// TIA Portal project "Banda_Asamblare" (V15.1)

(* hardware
DEVICE "S71500/ET200MP station_1"  S7-1500 station
   slot 0: "Rail_0"  Rack  6ES7 590-1***0-0AA0
   slot 1: "PLC_1"  CPU 1513-1 PN  6ES7 513-1AL02-0AB0  V2.6
      slot 3: "CPU display_1"  6ES7591-1AA00-0AA0
*)

// ===== PLC "PLC_1"  CPU 1513-1 PN =====

VAR_GLOBAL   // PLC tag table "Default tag table"
   "Clock_Byte" AT %MB0 : Byte;
   "Clock_10Hz" AT %M0.0 : Bool;
   "Clock_5Hz" AT %M0.1 : Bool;
   "Clock_2.5Hz" AT %M0.2 : Bool;
   "Clock_2Hz" AT %M0.3 : Bool;
   "Clock_1.25Hz" AT %M0.4 : Bool;
   "Clock_1Hz" AT %M0.5 : Bool;
   "Clock_0.625Hz" AT %M0.6 : Bool;
   "Clock_0.5Hz" AT %M0.7 : Bool;
END_VAR

DATA_BLOCK "Alarme"   // DB1
{ S7_Optimized_Access := 'TRUE' }
VERSION : 0.1
   VAR
      alarme_vect : Array[0..15] of Bool;
      alarme_gather : Word;
   END_VAR
BEGIN
END_DATA_BLOCK

DATA_BLOCK "Avarii"   // DB2
{ S7_Optimized_Access := 'TRUE' }
VERSION : 0.1
   VAR
      avarie_start : Bool;
      avarie_cuptor : Bool;
      avarie_aplatizor : Bool;
      avarie_forme : Bool;
      avarie_taiere : Bool;
      avarie_curatare : Bool;
      avarie_general : Bool;
      container1_plin : Bool;
      container2_plin : Bool;
      container3_plin : Bool;
      container_plin_general : Bool;
      limite_containere : Bool;
   END_VAR
BEGIN
END_DATA_BLOCK

DATA_BLOCK "Mecanisme"   // DB3
{ S7_Optimized_Access := 'TRUE' }
VERSION : 0.1
   VAR
      block_start : Bool;
      punere_block_material : Bool;
      cuptor : Bool;
      temperatura_cuptor : Real;
      "temperatura dorita la cuptor" : Real;
      temp_dorita_atinsa : Bool;
      aplatizor : Bool;
      forma : UInt;
      ajuns_la_forma1 : Bool;
      ajuns_la_forma2 : Bool;
      ajuns_la_forma3 : Bool;
      taiere1 : Bool;
      taiere2 : Bool;
      taiere3 : Bool;
      curatare1 : Bool;
      curatare2 : Bool;
      curatare3 : Bool;
      container_f1 : UInt;
      container_f2 : UInt;
      container_f3 : UInt;
      servo : UInt;
      limita_c1 : UInt;
      limita_c2 : UInt;
      limita_c3 : UInt;
      cond_cuptor : Bool;
   END_VAR
BEGIN
END_DATA_BLOCK

DATA_BLOCK "Butoane"   // DB4
{ S7_Optimized_Access := 'TRUE' }
VERSION : 0.1
   VAR
      btn_start : Bool;
      btn_esd : Bool;
      btn_stop : Bool;
      reset_esd : Bool;
      pornire : Bool;
      esd : Bool;
      "blocare_start_pe timer" : Bool;
      mentinere_timer_punere_material : Bool;
      "reset avarii" : Bool;
      timer_oprit : Bool;
      golire_c1 : Bool;
      golire_c2 : Bool;
      golire_c3 : Bool;
   END_VAR
BEGIN
END_DATA_BLOCK

DATA_BLOCK "Benzi"   // DB5
{ S7_Optimized_Access := 'TRUE' }
VERSION : 0.1
   VAR
      plecat_b1 : Bool;
      plecat_b2 : Bool;
      plecat_b3 : Bool;
      plecat_b41 : Bool;
      plecat_b42 : Bool;
      plecat_b43 : Bool;
      plecat_b51 : Bool;
      plecat_b52 : Bool;
      plecat_b53 : Bool;
      plecat_b61 : Bool;
      plecat_b62 : Bool;
      plecat_b63 : Bool;
   END_VAR
BEGIN
END_DATA_BLOCK

DATA_BLOCK "Comenzi_DB"   // DB7
{ S7_Optimized_Access := 'TRUE' }
VERSION : 0.1
// stored: InstanceOfName Comenzi
"Comenzi"
BEGIN
END_DATA_BLOCK

DATA_BLOCK "rising edges"   // DB9
{ S7_Optimized_Access := 'TRUE' }
VERSION : 0.1
   VAR
      re1 : Bool;
      re2 : Bool;
      re3 : Bool;
      re4 : Bool;
      re5 : Bool;
      re6 : Bool;
      re7 : Bool;
      re8 : Bool;
   END_VAR
BEGIN
END_DATA_BLOCK

DATA_BLOCK "Simulare_DB"   // DB13
{ S7_Optimized_Access := 'TRUE' }
VERSION : 0.1
// stored: InstanceOfName Simulare
"Simulare"
BEGIN
END_DATA_BLOCK

// folder: System blocks/Program resources

DATA_BLOCK "reset esd"   // DB6
{ S7_Optimized_Access := 'TRUE' }
AUTHOR : Simatic
FAMILY : IEC
NAME : IEC_TMR
VERSION : 1.0
// stored: InstanceOfName IEC_TIMER
"IEC_TIMER"
BEGIN
END_DATA_BLOCK

// folder: (top level)

FUNCTION_BLOCK "Simulare"   // FB1, LAD
{ S7_Optimized_Access := 'TRUE' }
VERSION : 0.1
   VAR_INPUT
      btn_pornire : Bool;
      b1_plecat : Bool;
      b2_plecat : Bool;
      b3_plecat : Bool;
      b41_plecat : Bool;
      b42_plecat : Bool;
      b43_plecat : Bool;
      b51_plecat : Bool;
      b52_plecat : Bool;
      b53_plecat : Bool;
      b61_plecat : Bool;
      b62_plecat : Bool;
      b63_plecat : Bool;
      cond_cuptor : Bool;
      forma : UInt;
   END_VAR
   VAR_OUTPUT
      cuptor_pornit : Bool;
      aplatizor_pornit : Bool;
      forma1 : Bool;
      forma2 : Bool;
      forma3 : Bool;
      taiere1 : Bool;
      taiere2 : Bool;
      taiere3 : Bool;
      curatare1 : Bool;
      curatare2 : Bool;
      curatare3 : Bool;
      container1 : UInt;
      container2 : UInt;
      container3 : UInt;
      servo : UInt;
   END_VAR
   VAR_IN_OUT
      pune_material : Bool;
      btn_golire1 : Bool;
      btn_golire2 : Bool;
      btn_golire3 : Bool;
      temp_cuptor : Real;
   END_VAR
   VAR
      re1 : Bool;
      re2 : Bool;
      re3 : Bool;
      re4 : Bool;
      re5 : Bool;
      "timer reset punere material" : TON_TIME;
      mentinere_timer_material : Bool;
      timer_aplatizare : TON_TIME;
      "tiimer forma" : TON_TIME;
      "timer taiere1" : TON_TIME;
      "timer taiere2" : TON_TIME;
      "timer taiere3" : TON_TIME;
      "timer curatare1" : TON_TIME;
      "timer curatare 2" : TON_TIME;
      "timer curatare 3" : TON_TIME;
      "reset golire1" : TON_TIME;
      "reset golire 2" : TON_TIME;
      "reset golire 3" : TON_TIME;
   END_VAR
   VAR_TEMP   // added for the SCL form of the ladder/FBD networks
      _w1 : Bool;
      _w2 : Bool;
      _w3 : Bool;
   END_VAR
BEGIN

REGION Network 1: pune un block de material pe banda
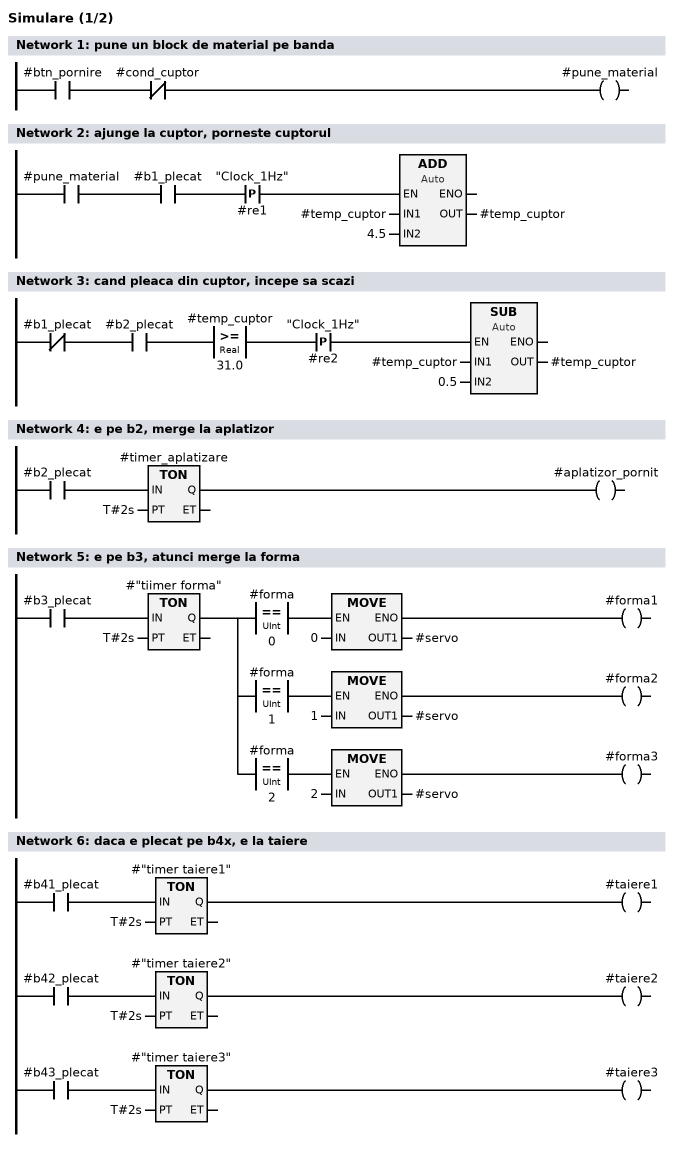
   RUNG wire#powerrail
      Contact( #btn_pornire )
      I_Contact( #cond_cuptor )
      Coil( #pune_material )
   END_RUNG
   // the same network as SCL:
   #pune_material := #btn_pornire AND NOT #cond_cuptor;
END_REGION

REGION Network 2: ajunge la cuptor, porneste cuptorul
   RUNG wire#powerrail
      Contact( #pune_material )
      Contact( #b1_plecat )
      P_Contact(operand := "Clock_1Hz", bit := #re1)
      Add(in1 := #temp_cuptor, in2 := 4.5, out => #temp_cuptor)
   END_RUNG
   // the same network as SCL:
   #_w1 := #pune_material AND #b1_plecat AND "Clock_1Hz" AND NOT #re1;   // rising edge of "Clock_1Hz"
   #re1 := "Clock_1Hz";
   IF #_w1 THEN #temp_cuptor := #temp_cuptor + 4.5; END_IF;
END_REGION

REGION Network 3: cand pleaca din cuptor, incepe sa scazi
   RUNG wire#powerrail
      I_Contact( #b1_plecat )
      Contact( #b2_plecat )
      { S7_Templates := "SrcType := Real" } GE_Contact(in1 := #temp_cuptor, in2 := 31.0)
      P_Contact(operand := "Clock_1Hz", bit := #re2)
      Sub(in1 := #temp_cuptor, in2 := 0.5, out => #temp_cuptor)
   END_RUNG
   // the same network as SCL:
   #_w1 := NOT #b1_plecat AND #b2_plecat AND (#temp_cuptor >= 31.0) AND "Clock_1Hz" AND NOT #re2;   // rising edge of "Clock_1Hz"
   #re2 := "Clock_1Hz";
   IF #_w1 THEN #temp_cuptor := #temp_cuptor - 0.5; END_IF;
END_REGION

REGION Network 4: e pe b2, merge la aplatizor
   #timer_aplatizare(IN := #b2_plecat, PT := T#2s);   // TON
   #aplatizor_pornit := #timer_aplatizare.Q;
END_REGION

REGION Network 5: e pe b3, atunci merge la forma
   #"tiimer forma"(IN := #b3_plecat, PT := T#2s);   // TON
   #_w1 := #"tiimer forma".Q AND (#forma = 0);
   IF #_w1 THEN #servo := 0; END_IF;
   #forma1 := #_w1;
   #_w2 := #"tiimer forma".Q AND (#forma = 1);
   IF #_w2 THEN #servo := 1; END_IF;
   #forma2 := #_w2;
   #_w3 := #"tiimer forma".Q AND (#forma = 2);
   IF #_w3 THEN #servo := 2; END_IF;
   #forma3 := #_w3;
END_REGION

REGION Network 6: daca e plecat pe b4x, e la taiere
   #"timer taiere1"(IN := #b41_plecat, PT := T#2s);   // TON
   #taiere1 := #"timer taiere1".Q;
   #"timer taiere2"(IN := #b42_plecat, PT := T#2s);   // TON
   #taiere2 := #"timer taiere2".Q;
   #"timer taiere3"(IN := #b43_plecat, PT := T#2s);   // TON
   #taiere3 := #"timer taiere3".Q;
END_REGION

REGION Network 7: daca e pe banda b5x, sa dea drumul la curatari
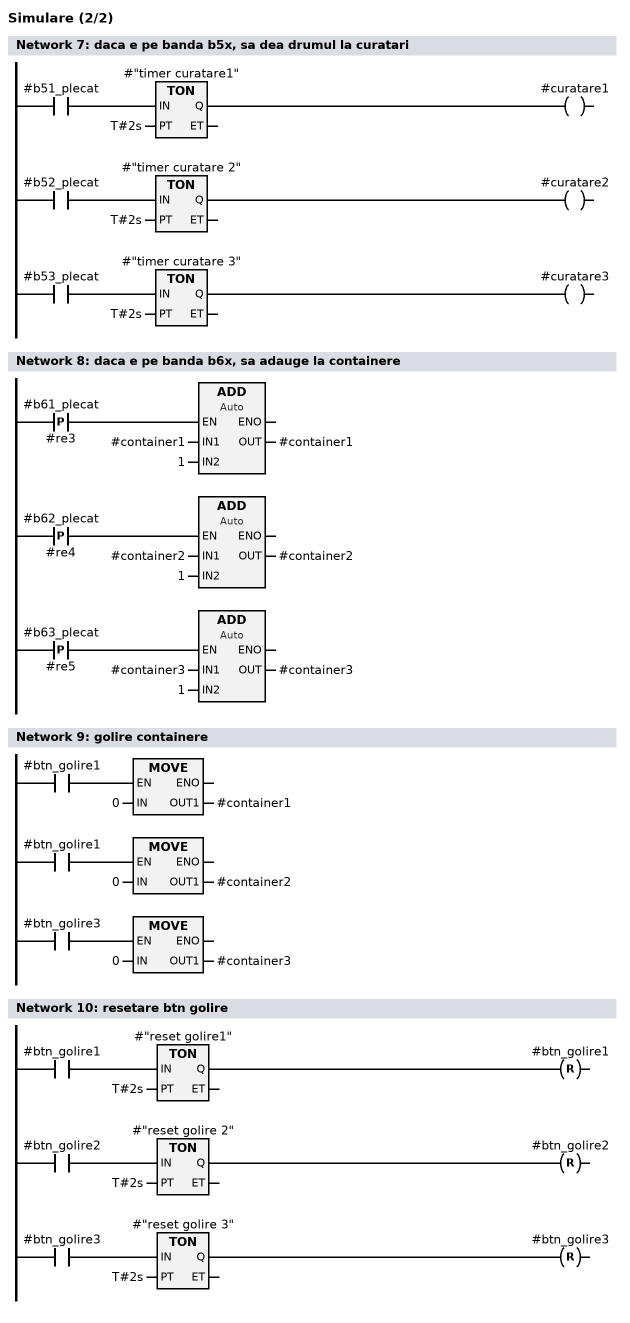
   #"timer curatare1"(IN := #b51_plecat, PT := T#2s);   // TON
   #curatare1 := #"timer curatare1".Q;
   #"timer curatare 2"(IN := #b52_plecat, PT := T#2s);   // TON
   #curatare2 := #"timer curatare 2".Q;
   #"timer curatare 3"(IN := #b53_plecat, PT := T#2s);   // TON
   #curatare3 := #"timer curatare 3".Q;
END_REGION

REGION Network 8: daca e pe banda b6x, sa adauge la containere
   RUNG wire#powerrail
      P_Contact(operand := #b61_plecat, bit := #re3)
      Add(in1 := #container1, in2 := 1, out => #container1)
   END_RUNG
   RUNG wire#powerrail
      P_Contact(operand := #b62_plecat, bit := #re4)
      Add(in1 := #container2, in2 := 1, out => #container2)
   END_RUNG
   RUNG wire#powerrail
      P_Contact(operand := #b63_plecat, bit := #re5)
      Add(in1 := #container3, in2 := 1, out => #container3)
   END_RUNG
   // the same network as SCL:
   #_w1 := #b61_plecat AND NOT #re3;   // rising edge of #b61_plecat
   #re3 := #b61_plecat;
   IF #_w1 THEN #container1 := #container1 + 1; END_IF;
   #_w2 := #b62_plecat AND NOT #re4;   // rising edge of #b62_plecat
   #re4 := #b62_plecat;
   IF #_w2 THEN #container2 := #container2 + 1; END_IF;
   #_w3 := #b63_plecat AND NOT #re5;   // rising edge of #b63_plecat
   #re5 := #b63_plecat;
   IF #_w3 THEN #container3 := #container3 + 1; END_IF;
END_REGION

REGION Network 9: golire containere
   RUNG wire#powerrail
      Contact( #btn_golire1 )
      Move(in := 0, out1 => #container1)
   END_RUNG
   RUNG wire#powerrail
      Contact( #btn_golire1 )
      Move(in := 0, out1 => #container2)
   END_RUNG
   RUNG wire#powerrail
      Contact( #btn_golire3 )
      Move(in := 0, out1 => #container3)
   END_RUNG
   // the same network as SCL:
   IF #btn_golire1 THEN
       #container1 := 0;
       #container2 := 0;
   END_IF;
   IF #btn_golire3 THEN #container3 := 0; END_IF;
END_REGION

REGION Network 10: resetare btn golire
   #"reset golire1"(IN := #btn_golire1, PT := T#2s);   // TON
   IF #"reset golire1".Q THEN #btn_golire1 := FALSE; END_IF;
   #"reset golire 2"(IN := #btn_golire2, PT := T#2s);   // TON
   IF #"reset golire 2".Q THEN #btn_golire2 := FALSE; END_IF;
   #"reset golire 3"(IN := #btn_golire3, PT := T#2s);   // TON
   IF #"reset golire 3".Q THEN #btn_golire3 := FALSE; END_IF;
END_REGION
END_FUNCTION_BLOCK

FUNCTION_BLOCK "Comenzi"   // FB2, LAD
{ S7_Optimized_Access := 'TRUE' }
VERSION : 0.1
   VAR_INPUT
      temp_cuptor : Real;
      temp_dorita : Real;
      pune_material : Bool;
      aplatizor_pornit : Bool;
      forma1 : Bool;
      forma2 : Bool;
      forma3 : Bool;
      taiere1 : Bool;
      taiere2 : Bool;
      taiere3 : Bool;
      curatare1 : Bool;
      curatare2 : Bool;
      curatare3 : Bool;
   END_VAR
   VAR_OUTPUT
      b1_plecat : Bool;
      b2_plecat : Bool;
      b3_plecat : Bool;
      b41_plecat : Bool;
      b42_plecat : Bool;
      b43_plecat : Bool;
      b51_plecat : Bool;
      b52_plecat : Bool;
      b53_plecat : Bool;
      b61_plecat : Bool;
      b62_plecat : Bool;
      b63_plecat : Bool;
      cond_cuptor : Bool;
   END_VAR
   VAR
      "timer plecare b1" : TON_TIME;
      incc : Int;
      edg : Bool;
   END_VAR
BEGIN

REGION Network 1: pleaca spre cuptor
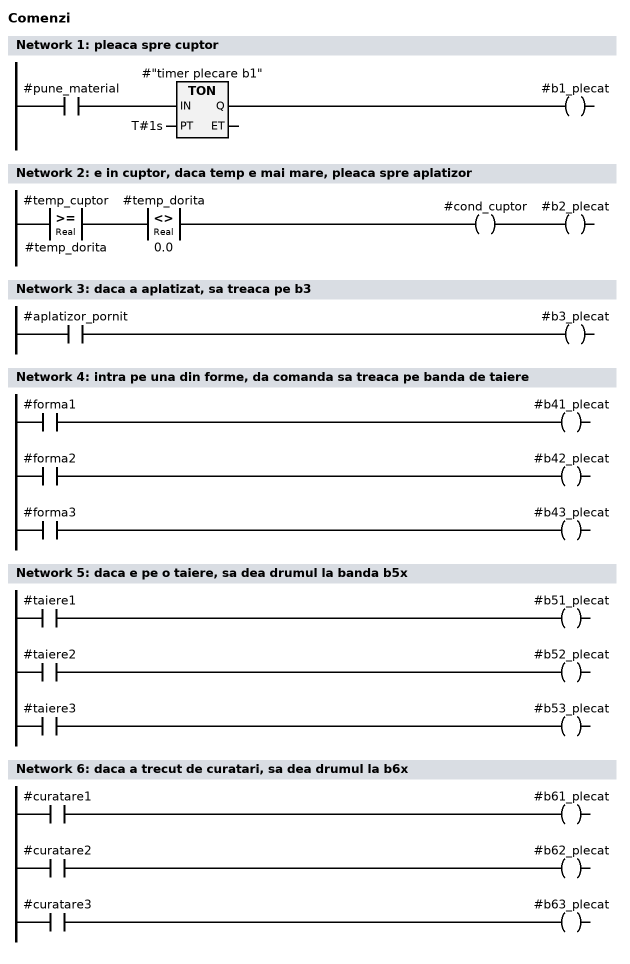
   #"timer plecare b1"(IN := #pune_material, PT := T#1s);   // TON
   #b1_plecat := #"timer plecare b1".Q;
END_REGION

REGION Network 2: e in cuptor, daca temp e mai mare, pleaca spre aplatizor
   RUNG wire#powerrail
      { S7_Templates := "SrcType := Real" } GE_Contact(in1 := #temp_cuptor, in2 := #temp_dorita)
      { S7_Templates := "SrcType := Real" } NE_Contact(in1 := #temp_dorita, in2 := 0.0)
      Coil( #cond_cuptor )
      Coil( #b2_plecat )
   END_RUNG
   // the same network as SCL:
   #cond_cuptor := (#temp_cuptor >= #temp_dorita) AND (#temp_dorita <> 0.0);
   #b2_plecat := #cond_cuptor;
END_REGION

REGION Network 3: daca a aplatizat, sa treaca pe b3
   RUNG wire#powerrail
      Contact( #aplatizor_pornit )
      Coil( #b3_plecat )
   END_RUNG
   // the same network as SCL:
   #b3_plecat := #aplatizor_pornit;
END_REGION

REGION Network 4: intra pe una din forme, da comanda sa treaca pe banda de taiere
   RUNG wire#powerrail
      Contact( #forma1 )
      Coil( #b41_plecat )
   END_RUNG
   RUNG wire#powerrail
      Contact( #forma2 )
      Coil( #b42_plecat )
   END_RUNG
   RUNG wire#powerrail
      Contact( #forma3 )
      Coil( #b43_plecat )
   END_RUNG
   // the same network as SCL:
   #b41_plecat := #forma1;
   #b42_plecat := #forma2;
   #b43_plecat := #forma3;
END_REGION

REGION Network 5: daca e pe o taiere, sa dea drumul la banda b5x
   RUNG wire#powerrail
      Contact( #taiere1 )
      Coil( #b51_plecat )
   END_RUNG
   RUNG wire#powerrail
      Contact( #taiere2 )
      Coil( #b52_plecat )
   END_RUNG
   RUNG wire#powerrail
      Contact( #taiere3 )
      Coil( #b53_plecat )
   END_RUNG
   // the same network as SCL:
   #b51_plecat := #taiere1;
   #b52_plecat := #taiere2;
   #b53_plecat := #taiere3;
END_REGION

REGION Network 6: daca a trecut de curatari, sa dea drumul la b6x
   RUNG wire#powerrail
      Contact( #curatare1 )
      Coil( #b61_plecat )
   END_RUNG
   RUNG wire#powerrail
      Contact( #curatare2 )
      Coil( #b62_plecat )
   END_RUNG
   RUNG wire#powerrail
      Contact( #curatare3 )
      Coil( #b63_plecat )
   END_RUNG
   // the same network as SCL:
   #b61_plecat := #curatare1;
   #b62_plecat := #curatare2;
   #b63_plecat := #curatare3;
END_REGION
END_FUNCTION_BLOCK

ORGANIZATION_BLOCK "Main"   // OB1, LAD, ProgramCycle
TITLE = "Main Program Sweep (Cycle)"
{ S7_Optimized_Access := 'TRUE' }
VERSION : 0.1
   VAR_INPUT
      Initial_Call : Bool;   // Initial call of this OB
      Remanence : Bool;   // =True, if remanent data are available
   END_VAR
BEGIN

REGION Network 1: buton start
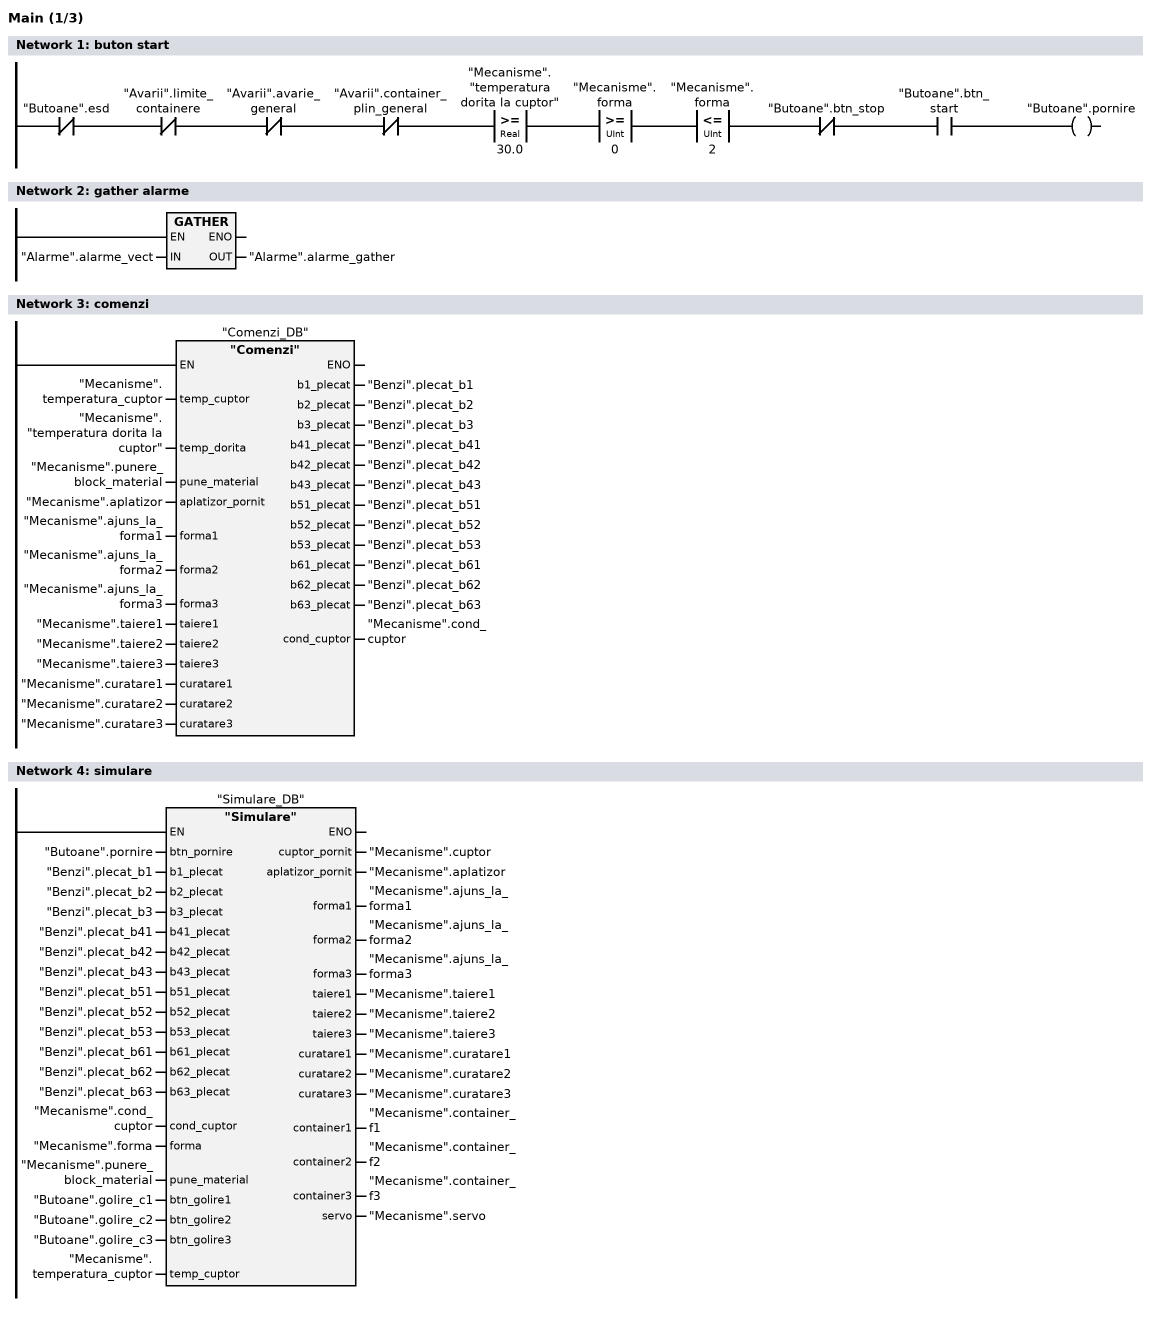
   RUNG wire#powerrail
      I_Contact( "Butoane".esd )
      I_Contact( "Avarii".limite_containere )
      I_Contact( "Avarii".avarie_general )
      I_Contact( "Avarii".container_plin_general )
      { S7_Templates := "SrcType := Real" } GE_Contact(in1 := "Mecanisme"."temperatura dorita la cuptor", in2 := 30.0)
      { S7_Templates := "SrcType := UInt" } GE_Contact(in1 := "Mecanisme".forma, in2 := 0)
      { S7_Templates := "SrcType := UInt" } LE_Contact(in1 := "Mecanisme".forma, in2 := 2)
      I_Contact( "Butoane".btn_stop )
      Contact( "Butoane".btn_start )
      Coil( "Butoane".pornire )
   END_RUNG
   // the same network as SCL:
   "Butoane".pornire := NOT "Butoane".esd AND NOT "Avarii".limite_containere AND NOT "Avarii".avarie_general AND NOT "Avarii".container_plin_general AND ("Mecanisme"."temperatura dorita la cuptor" >= 30.0) AND ("Mecanisme".forma >= 0) AND ("Mecanisme".forma <= 2) AND NOT "Butoane".btn_stop AND "Butoane".btn_start;
END_REGION

REGION Network 2: gather alarme
   GATHER(IN := "Alarme".alarme_vect, OUT => "Alarme".alarme_gather);
END_REGION

REGION Network 3: comenzi
   RUNG wire#powerrail
      "Comenzi_DB"(temp_cuptor := "Mecanisme".temperatura_cuptor, temp_dorita := "Mecanisme"."temperatura dorita la cuptor", pune_material := "Mecanisme".punere_block_material, aplatizor_pornit := "Mecanisme".aplatizor, forma1 := "Mecanisme".ajuns_la_forma1, forma2 := "Mecanisme".ajuns_la_forma2, forma3 := "Mecanisme".ajuns_la_forma3, taiere1 := "Mecanisme".taiere1, taiere2 := "Mecanisme".taiere2, taiere3 := "Mecanisme".taiere3, curatare1 := "Mecanisme".curatare1, curatare2 := "Mecanisme".curatare2, curatare3 := "Mecanisme".curatare3, b1_plecat => "Benzi".plecat_b1, b2_plecat => "Benzi".plecat_b2, b3_plecat => "Benzi".plecat_b3, b41_plecat => "Benzi".plecat_b41, b42_plecat => "Benzi".plecat_b42, b43_plecat => "Benzi".plecat_b43, b51_plecat => "Benzi".plecat_b51, b52_plecat => "Benzi".plecat_b52, b53_plecat => "Benzi".plecat_b53, b61_plecat => "Benzi".plecat_b61, b62_plecat => "Benzi".plecat_b62, b63_plecat => "Benzi".plecat_b63, cond_cuptor => "Mecanisme".cond_cuptor)
   END_RUNG
   // the same network as SCL:
   "Comenzi_DB"(temp_cuptor := "Mecanisme".temperatura_cuptor,   // "Comenzi"
                temp_dorita := "Mecanisme"."temperatura dorita la cuptor",
                pune_material := "Mecanisme".punere_block_material,
                aplatizor_pornit := "Mecanisme".aplatizor,
                forma1 := "Mecanisme".ajuns_la_forma1,
                forma2 := "Mecanisme".ajuns_la_forma2,
                forma3 := "Mecanisme".ajuns_la_forma3,
                taiere1 := "Mecanisme".taiere1,
                taiere2 := "Mecanisme".taiere2,
                taiere3 := "Mecanisme".taiere3,
                curatare1 := "Mecanisme".curatare1,
                curatare2 := "Mecanisme".curatare2,
                curatare3 := "Mecanisme".curatare3,
                b1_plecat => "Benzi".plecat_b1,
                b2_plecat => "Benzi".plecat_b2,
                b3_plecat => "Benzi".plecat_b3,
                b41_plecat => "Benzi".plecat_b41,
                b42_plecat => "Benzi".plecat_b42,
                b43_plecat => "Benzi".plecat_b43,
                b51_plecat => "Benzi".plecat_b51,
                b52_plecat => "Benzi".plecat_b52,
                b53_plecat => "Benzi".plecat_b53,
                b61_plecat => "Benzi".plecat_b61,
                b62_plecat => "Benzi".plecat_b62,
                b63_plecat => "Benzi".plecat_b63,
                cond_cuptor => "Mecanisme".cond_cuptor);
END_REGION

REGION Network 4: simulare
   RUNG wire#powerrail
      "Simulare_DB"(btn_pornire := "Butoane".pornire, b1_plecat := "Benzi".plecat_b1, b2_plecat := "Benzi".plecat_b2, b3_plecat := "Benzi".plecat_b3, b41_plecat := "Benzi".plecat_b41, b42_plecat := "Benzi".plecat_b42, b43_plecat := "Benzi".plecat_b43, b51_plecat := "Benzi".plecat_b51, b52_plecat := "Benzi".plecat_b52, b53_plecat := "Benzi".plecat_b53, b61_plecat := "Benzi".plecat_b61, b62_plecat := "Benzi".plecat_b62, b63_plecat := "Benzi".plecat_b63, cond_cuptor := "Mecanisme".cond_cuptor, forma := "Mecanisme".forma, btn_golire1 := "Butoane".golire_c1, btn_golire2 := "Butoane".golire_c2, btn_golire3 := "Butoane".golire_c3, pune_material := "Mecanisme".punere_block_material, temp_cuptor := "Mecanisme".temperatura_cuptor, cuptor_pornit => "Mecanisme".cuptor, aplatizor_pornit => "Mecanisme".aplatizor, forma1 => "Mecanisme".ajuns_la_forma1, forma2 => "Mecanisme".ajuns_la_forma2, forma3 => "Mecanisme".ajuns_la_forma3, taiere1 => "Mecanisme".taiere1, taiere2 => "Mecanisme".taiere2, taiere3 => "Mecanisme".taiere3, curatare1 => "Mecanisme".curatare1, curatare2 => "Mecanisme".curatare2, curatare3 => "Mecanisme".curatare3, container1 => "Mecanisme".container_f1, container2 => "Mecanisme".container_f2, container3 => "Mecanisme".container_f3, servo => "Mecanisme".servo)
   END_RUNG
   // the same network as SCL:
   "Simulare_DB"(btn_pornire := "Butoane".pornire,   // "Simulare"
                 b1_plecat := "Benzi".plecat_b1,
                 b2_plecat := "Benzi".plecat_b2,
                 b3_plecat := "Benzi".plecat_b3,
                 b41_plecat := "Benzi".plecat_b41,
                 b42_plecat := "Benzi".plecat_b42,
                 b43_plecat := "Benzi".plecat_b43,
                 b51_plecat := "Benzi".plecat_b51,
                 b52_plecat := "Benzi".plecat_b52,
                 b53_plecat := "Benzi".plecat_b53,
                 b61_plecat := "Benzi".plecat_b61,
                 b62_plecat := "Benzi".plecat_b62,
                 b63_plecat := "Benzi".plecat_b63,
                 cond_cuptor := "Mecanisme".cond_cuptor,
                 forma := "Mecanisme".forma,
                 pune_material := "Mecanisme".punere_block_material,
                 btn_golire1 := "Butoane".golire_c1,
                 btn_golire2 := "Butoane".golire_c2,
                 btn_golire3 := "Butoane".golire_c3,
                 temp_cuptor := "Mecanisme".temperatura_cuptor,
                 cuptor_pornit => "Mecanisme".cuptor,
                 aplatizor_pornit => "Mecanisme".aplatizor,
                 forma1 => "Mecanisme".ajuns_la_forma1,
                 forma2 => "Mecanisme".ajuns_la_forma2,
                 forma3 => "Mecanisme".ajuns_la_forma3,
                 taiere1 => "Mecanisme".taiere1,
                 taiere2 => "Mecanisme".taiere2,
                 taiere3 => "Mecanisme".taiere3,
                 curatare1 => "Mecanisme".curatare1,
                 curatare2 => "Mecanisme".curatare2,
                 curatare3 => "Mecanisme".curatare3,
                 container1 => "Mecanisme".container_f1,
                 container2 => "Mecanisme".container_f2,
                 container3 => "Mecanisme".container_f3,
                 servo => "Mecanisme".servo);
END_REGION

REGION Network 5: esd
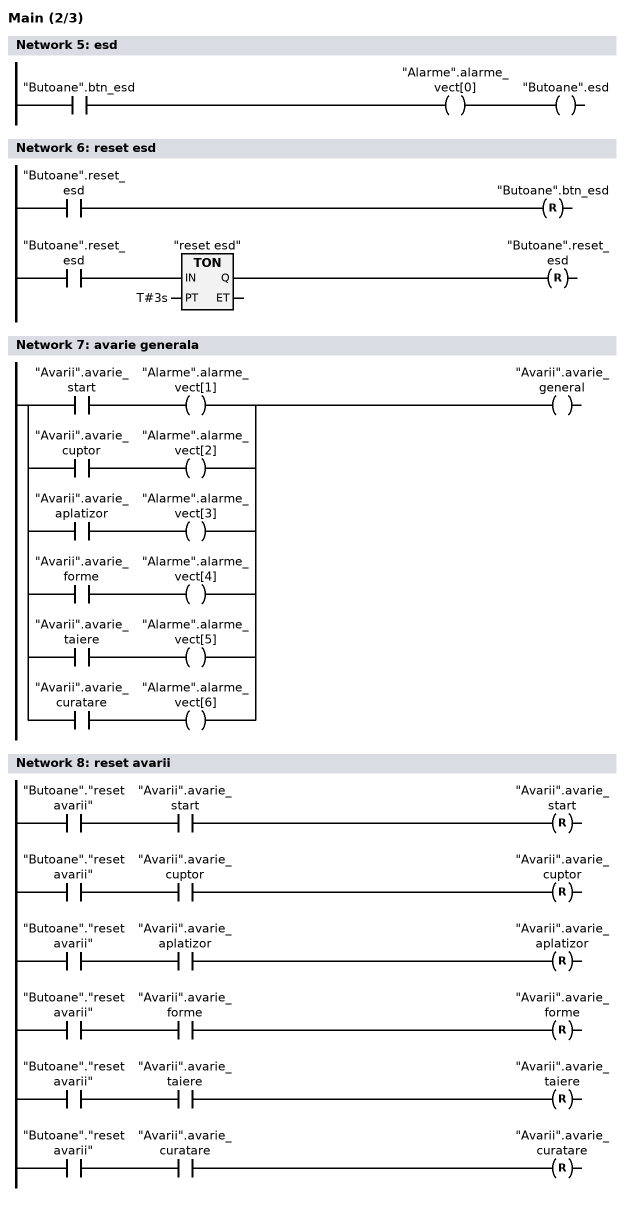
   RUNG wire#powerrail
      Contact( "Butoane".btn_esd )
      Coil( "Alarme".alarme_vect[0] )
      Coil( "Butoane".esd )
   END_RUNG
   // the same network as SCL:
   "Alarme".alarme_vect[0] := "Butoane".btn_esd;
   "Butoane".esd := "Butoane".btn_esd;
END_REGION

REGION Network 6: reset esd
   IF "Butoane".reset_esd THEN "Butoane".btn_esd := FALSE; END_IF;
   "reset esd".TON(IN := "Butoane".reset_esd, PT := T#3s);
   IF "reset esd".Q THEN "Butoane".reset_esd := FALSE; END_IF;
END_REGION

REGION Network 7: avarie generala
   RUNG wire#powerrail
      Contact( "Avarii".avarie_start )
      Coil( "Alarme".alarme_vect[1] )
      wire#w1
      Coil( "Avarii".avarie_general )
   END_RUNG
   RUNG wire#powerrail
      Contact( "Avarii".avarie_cuptor )
      Coil( "Alarme".alarme_vect[2] )
   END_RUNG wire#w1
   RUNG wire#powerrail
      Contact( "Avarii".avarie_aplatizor )
      Coil( "Alarme".alarme_vect[3] )
   END_RUNG wire#w1
   RUNG wire#powerrail
      Contact( "Avarii".avarie_forme )
      Coil( "Alarme".alarme_vect[4] )
   END_RUNG wire#w1
   RUNG wire#powerrail
      Contact( "Avarii".avarie_taiere )
      Coil( "Alarme".alarme_vect[5] )
   END_RUNG wire#w1
   RUNG wire#powerrail
      Contact( "Avarii".avarie_curatare )
      Coil( "Alarme".alarme_vect[6] )
   END_RUNG wire#w1
   // the same network as SCL:
   "Alarme".alarme_vect[1] := "Avarii".avarie_start;
   "Alarme".alarme_vect[2] := "Avarii".avarie_cuptor;
   "Alarme".alarme_vect[3] := "Avarii".avarie_aplatizor;
   "Alarme".alarme_vect[4] := "Avarii".avarie_forme;
   "Alarme".alarme_vect[5] := "Avarii".avarie_taiere;
   "Alarme".alarme_vect[6] := "Avarii".avarie_curatare;
   "Avarii".avarie_general := "Avarii".avarie_start OR "Avarii".avarie_cuptor OR "Avarii".avarie_aplatizor OR "Avarii".avarie_forme OR "Avarii".avarie_taiere OR "Avarii".avarie_curatare;
END_REGION

REGION Network 8: reset avarii
   RUNG wire#powerrail
      Contact( "Butoane"."reset avarii" )
      Contact( "Avarii".avarie_start )
      R_Coil( "Avarii".avarie_start )
   END_RUNG
   RUNG wire#powerrail
      Contact( "Butoane"."reset avarii" )
      Contact( "Avarii".avarie_cuptor )
      R_Coil( "Avarii".avarie_cuptor )
   END_RUNG
   RUNG wire#powerrail
      Contact( "Butoane"."reset avarii" )
      Contact( "Avarii".avarie_aplatizor )
      R_Coil( "Avarii".avarie_aplatizor )
   END_RUNG
   RUNG wire#powerrail
      Contact( "Butoane"."reset avarii" )
      Contact( "Avarii".avarie_forme )
      R_Coil( "Avarii".avarie_forme )
   END_RUNG
   RUNG wire#powerrail
      Contact( "Butoane"."reset avarii" )
      Contact( "Avarii".avarie_taiere )
      R_Coil( "Avarii".avarie_taiere )
   END_RUNG
   RUNG wire#powerrail
      Contact( "Butoane"."reset avarii" )
      Contact( "Avarii".avarie_curatare )
      R_Coil( "Avarii".avarie_curatare )
   END_RUNG
   // the same network as SCL:
   IF "Butoane"."reset avarii" AND "Avarii".avarie_start THEN "Avarii".avarie_start := FALSE; END_IF;
   IF "Butoane"."reset avarii" AND "Avarii".avarie_cuptor THEN "Avarii".avarie_cuptor := FALSE; END_IF;
   IF "Butoane"."reset avarii" AND "Avarii".avarie_aplatizor THEN "Avarii".avarie_aplatizor := FALSE; END_IF;
   IF "Butoane"."reset avarii" AND "Avarii".avarie_forme THEN "Avarii".avarie_forme := FALSE; END_IF;
   IF "Butoane"."reset avarii" AND "Avarii".avarie_taiere THEN "Avarii".avarie_taiere := FALSE; END_IF;
   IF "Butoane"."reset avarii" AND "Avarii".avarie_curatare THEN "Avarii".avarie_curatare := FALSE; END_IF;
END_REGION

REGION Network 9: container plin general
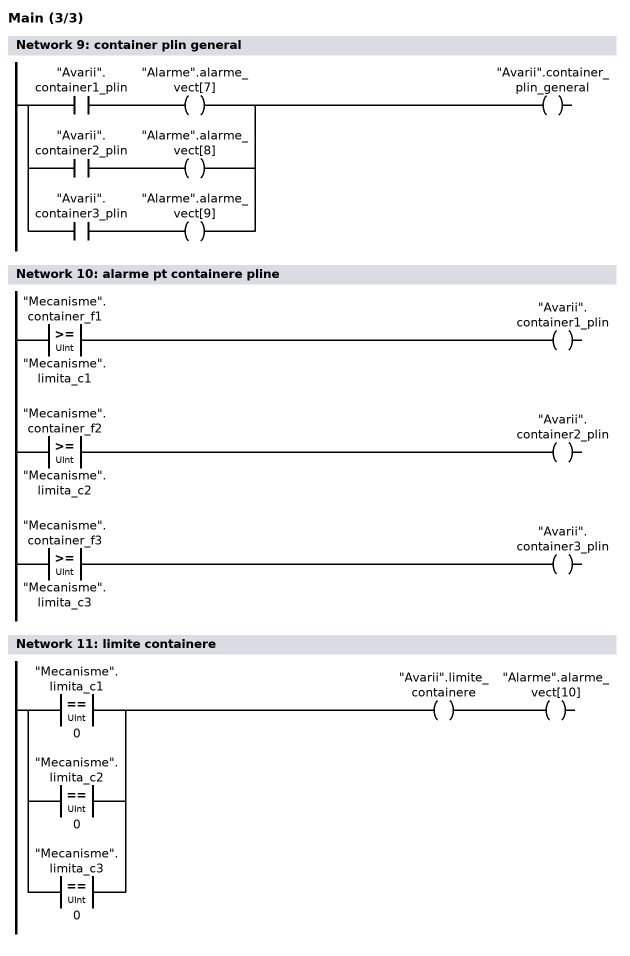
   RUNG wire#powerrail
      Contact( "Avarii".container1_plin )
      Coil( "Alarme".alarme_vect[7] )
      wire#w1
      Coil( "Avarii".container_plin_general )
   END_RUNG
   RUNG wire#powerrail
      Contact( "Avarii".container2_plin )
      Coil( "Alarme".alarme_vect[8] )
   END_RUNG wire#w1
   RUNG wire#powerrail
      Contact( "Avarii".container3_plin )
      Coil( "Alarme".alarme_vect[9] )
   END_RUNG wire#w1
   // the same network as SCL:
   "Alarme".alarme_vect[7] := "Avarii".container1_plin;
   "Alarme".alarme_vect[8] := "Avarii".container2_plin;
   "Alarme".alarme_vect[9] := "Avarii".container3_plin;
   "Avarii".container_plin_general := "Avarii".container1_plin OR "Avarii".container2_plin OR "Avarii".container3_plin;
END_REGION

REGION Network 10: alarme pt containere pline
   RUNG wire#powerrail
      { S7_Templates := "SrcType := UInt" } GE_Contact(in1 := "Mecanisme".container_f1, in2 := "Mecanisme".limita_c1)
      Coil( "Avarii".container1_plin )
   END_RUNG
   RUNG wire#powerrail
      { S7_Templates := "SrcType := UInt" } GE_Contact(in1 := "Mecanisme".container_f2, in2 := "Mecanisme".limita_c2)
      Coil( "Avarii".container2_plin )
   END_RUNG
   RUNG wire#powerrail
      { S7_Templates := "SrcType := UInt" } GE_Contact(in1 := "Mecanisme".container_f3, in2 := "Mecanisme".limita_c3)
      Coil( "Avarii".container3_plin )
   END_RUNG
   // the same network as SCL:
   "Avarii".container1_plin := "Mecanisme".container_f1 >= "Mecanisme".limita_c1;
   "Avarii".container2_plin := "Mecanisme".container_f2 >= "Mecanisme".limita_c2;
   "Avarii".container3_plin := "Mecanisme".container_f3 >= "Mecanisme".limita_c3;
END_REGION

REGION Network 11: limite containere
   RUNG wire#powerrail
      { S7_Templates := "SrcType := UInt" } EQ_Contact(in1 := "Mecanisme".limita_c1, in2 := 0)
      wire#w1
      Coil( "Avarii".limite_containere )
      Coil( "Alarme".alarme_vect[10] )
   END_RUNG
   RUNG wire#powerrail
      { S7_Templates := "SrcType := UInt" } EQ_Contact(in1 := "Mecanisme".limita_c2, in2 := 0)
   END_RUNG wire#w1
   RUNG wire#powerrail
      { S7_Templates := "SrcType := UInt" } EQ_Contact(in1 := "Mecanisme".limita_c3, in2 := 0)
   END_RUNG wire#w1
   // the same network as SCL:
   "Avarii".limite_containere := ("Mecanisme".limita_c1 = 0) OR ("Mecanisme".limita_c2 = 0) OR ("Mecanisme".limita_c3 = 0);
   "Alarme".alarme_vect[10] := "Avarii".limite_containere;
END_REGION
END_ORGANIZATION_BLOCK